Fanuc TP program (LS listing): _VIS_TEST.LS

/PROG  _VIS_TEST
/ATTR
OWNER		= MNEDITOR;
COMMENT		= "";
PROG_SIZE	= 708;
CREATE		= DATE 23-09-08  TIME 15:15:00;
MODIFIED	= DATE 23-09-08  TIME 15:22:14;
FILE_NAME	= ;
VERSION		= 0;
LINE_COUNT	= 10;
MEMORY_SIZE	= 1172;
PROTECT		= READ_WRITE;
TCD:  STACK_SIZE	= 0,
      TASK_PRIORITY	= 50,
      TIME_SLICE	= 0,
      BUSY_LAMP_OFF	= 0,
      ABORT_REQUEST	= 0,
      PAUSE_REQUEST	= 0;
DEFAULT_GROUP	= 1,*,*,*,*;
CONTROL_CODE	= 00000000 00000000;
LOCAL_REGISTERS	= 0,0,0;
/APPL
/APPL

AUTO_SINGULARITY_HEADER;
  ENABLE_SINGULARITY_AVOIDANCE   : FALSE;

PLTZ_MODE_HEADER;
 PLTZ_MODE_ENABLE   : FALSE;
 J4TURN  : ZERORAD;
 ORIENT  : DOWNWARDS;
/MN
   1:J P[1] 100% FINE    ;
   2:   ;
   3:  WAIT   1.00(sec) ;
   4:   ;
   5:  VISION RUN_FIND 'FINDRIGHTBOX'    ;
   6:  VISION GET_OFFSET 'FINDRIGHTBOX' VR[1] JMP LBL[99] ;
   7:J P[2] 100% FINE VOFFSET,VR[1] Offset,PR[65:50mm Z]    ;
   8:L P[2] 750mm/sec FINE VOFFSET,VR[1]    ;
   9:   ;
  10:  LBL[99] ;
/POS
P[1]{
   GP1:
	UF : 1, UT : 1,		CONFIG : 'N U T, 0, 0, 0',
	X =   634.375610  mm,	Y =   841.557007  mm,	Z =  1118.510254  mm,
	W =  -178.183594 deg,	P =     -.487492 deg,	R =   -89.865776 deg
};
P[2]{
   GP1:
	UF : 1, UT : 1,		CONFIG : 'N U T, 0, 0, 0',
	X =   -63.198303  mm,	Y =    73.658264  mm,	Z =   665.400452  mm,
	W =  -178.178925 deg,	P =     -.483090 deg,	R =    90.310623 deg
};
/END
